// SIMATIC S7-200 project (STEP 7-Micro/WIN), CPU 224 REL 01.22

ORGANIZATION_BLOCK MAIN:OB1
TITLE= 
// PROGRAM COMMENTS
// Press F1 for help and example program
//  
// 
BEGIN
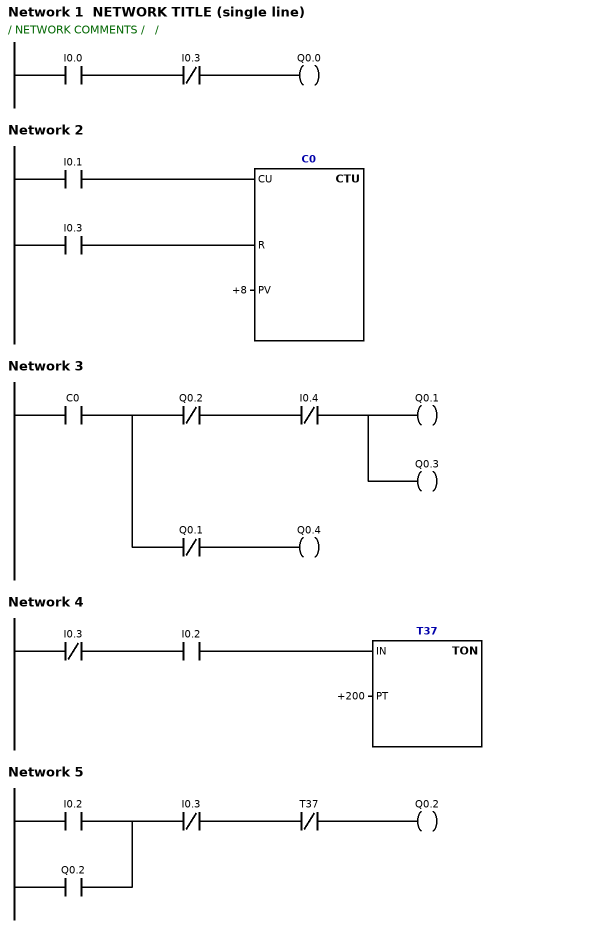
Network 1 // NETWORK TITLE (single line)
//  
// NETWORK COMMENTS
//  
// 
// (network saved uncompiled; LAD cells follow)
// row 0: c0 -| |- I0.0  c1 -|/|- I0.3  c2 -( ) Q0.0
Network 2
LD     I0.1
LD     I0.3
CTU    C0, +8
Network 3
LD     C0
LPS
AN     Q0.2
AN     I0.4
=      Q0.1
=      Q0.3
LPP
AN     Q0.1
=      Q0.4
Network 4
LDN    I0.3
A      I0.2
TON    T37, +200
Network 5
LD     I0.2
O      Q0.2
AN     I0.3
AN     T37
=      Q0.2
END_ORGANIZATION_BLOCK
